// Mitsubishi GX Works2 project: PLC_GROUP17   PLC: FX3G

// global labels: Global1
VAR_GLOBAL
  work_day AT X007 : BOOL;
  active_day AT Y007 : BOOL;
  emergency_sw AT X005 : BOOL;
  enter_inventory AT X010 : BOOL;
  chocolate_stock AT D1100 : REAL;
  input_chocolate AT D1110 : REAL;
  nuts_stock AT D1120 : REAL;
  input_nuts AT D1130 : REAL;
  pistachio_stock AT D1140 : REAL;
  input_pistachio AT D1150 : REAL;
  kadaif_stock AT D1160 : REAL;
  input_kadaif AT D1170 : REAL;
  input_sw AT M0 : BOOL;
  check_stock AT M1 : BOOL;
  finish_one_pack AT Y005 : BOOL;
END_VAR
VAR_GLOBAL CONSTANT
  min_chocolate_stock : REAL := 400.0;
  min_nuts_stock : REAL := 100.0;
  min_pistachio : REAL := 120.0;
  min_kadaif_stock : REAL := 60.0;
END_VAR
VAR_GLOBAL
  chack_chocolate AT M2 : BOOL;
  check_choco AT M2 : BOOL;
  check_nuts AT M3 : BOOL;
  check_pist AT M4 : BOOL;
  check_kadaif AT M5 : BOOL;
  start_melting AT X001 : BOOL;
  melting_light AT Y001 : BOOL;
  sensor_45 AT X002 : BOOL;
END_VAR
VAR_GLOBAL CONSTANT
  choco_amount : REAL := 400.0;
END_VAR
VAR_GLOBAL
  location_sensor AT X003 : BOOL;
  casting_light AT Y002 : BOOL;
  casting_timer AT TC200 : BOOL;
END_VAR
VAR_GLOBAL CONSTANT
  cast_time : INT := 400;
END_VAR
VAR_GLOBAL
  end_casting AT TS200 : BOOL;
  end_cast_light AT M6 : BOOL;
  sample_type AT X004 : BOOL;
  analog_input1 AT D8280 : INT;
  save_analog_input AT D1180 : REAL;
END_VAR
VAR_GLOBAL CONSTANT
  max_for_mix_nuts : REAL := 5.0;
END_VAR
VAR_GLOBAL
  mix_nuts_approved AT M7 : BOOL;
  transfer_light AT M6 : BOOL;
END_VAR
VAR_GLOBAL CONSTANT
  const400 : REAL := 400.0;
  const100 : REAL := 100.0;
END_VAR
VAR_GLOBAL
  mix_dubai_approved AT M8 : BOOL;
END_VAR
VAR_GLOBAL CONSTANT
  const60 : REAL := 60.0;
  const120 : REAL := 120.0;
  const20 : REAL := 20.0;
END_VAR
VAR_GLOBAL
  start_filling AT M9 : BOOL;
  timer_5_sec AT TC210 : BOOL;
END_VAR
VAR_GLOBAL CONSTANT
  filling_time : INT := 500;
END_VAR
VAR_GLOBAL
  filling_timer AT TS210 : BOOL;
  blink1 AT TC1 : BOOL;
END_VAR
VAR_GLOBAL CONSTANT
  blink1_time : INT := 10;
END_VAR
VAR_GLOBAL
  blink2 AT TC11 : BOOL;
END_VAR
VAR_GLOBAL CONSTANT
  blink_time : INT := 5;
END_VAR
VAR_GLOBAL
  blink_timer2 AT TS11 : BOOL;
  blink_light AT M10 : BOOL;
  blink_light1 AT Y003 : BOOL;
  blink_timer1 AT TS1 : BOOL;
  blink_light2 AT Y004 : BOOL;
  start_kirur AT X006 : BOOL;
  kirur_timer AT TC21 : BOOL;
END_VAR
VAR_GLOBAL CONSTANT
  kirur_time : INT := 30;
END_VAR
VAR_GLOBAL
  end_kirur AT TS21 : BOOL;
  kirur_light AT Y006 : BOOL;
  pack_table AT X000 : BOOL;
  table_counter AT CC0 : BOOL;
END_VAR
VAR_GLOBAL CONSTANT
  const4 : INT := 4;
END_VAR
VAR_GLOBAL
  pact_table_light AT Y005 : BOOL;
  end_full_package AT CS0 : BOOL;
  storage AT D1190 : REAL;
END_VAR
VAR_GLOBAL CONSTANT
  const1 : REAL := 1.0;
  const10 : INT := 10;
END_VAR
VAR_GLOBAL
  output AT D8282 : INT;
  reset_light AT M11 : BOOL;
  hold AT M12 : BOOL;
  hold2 AT M13 : BOOL;
  hold3 AT M14 : BOOL;
END_VAR
VAR_GLOBAL CONSTANT
  const40 : REAL := 40.0;
END_VAR
VAR_GLOBAL
  reset_storage_light AT M15 : BOOL;
END_VAR
VAR_GLOBAL CONSTANT
  const0 : REAL;
  const00 : INT;
END_VAR
VAR_GLOBAL
  which_mix AT M16 : BOOL;
  choco_sub_light AT M17 : BOOL;
END_VAR

// task Task_01 (event TRUE, interval 0, priority 31): POU_01

PROGRAM POU_01
(* structured ladder/FBD written out as ST: instructions are called as NAME(EN, inputs, outputs); _pN, _eN, _tN stand for wires *)
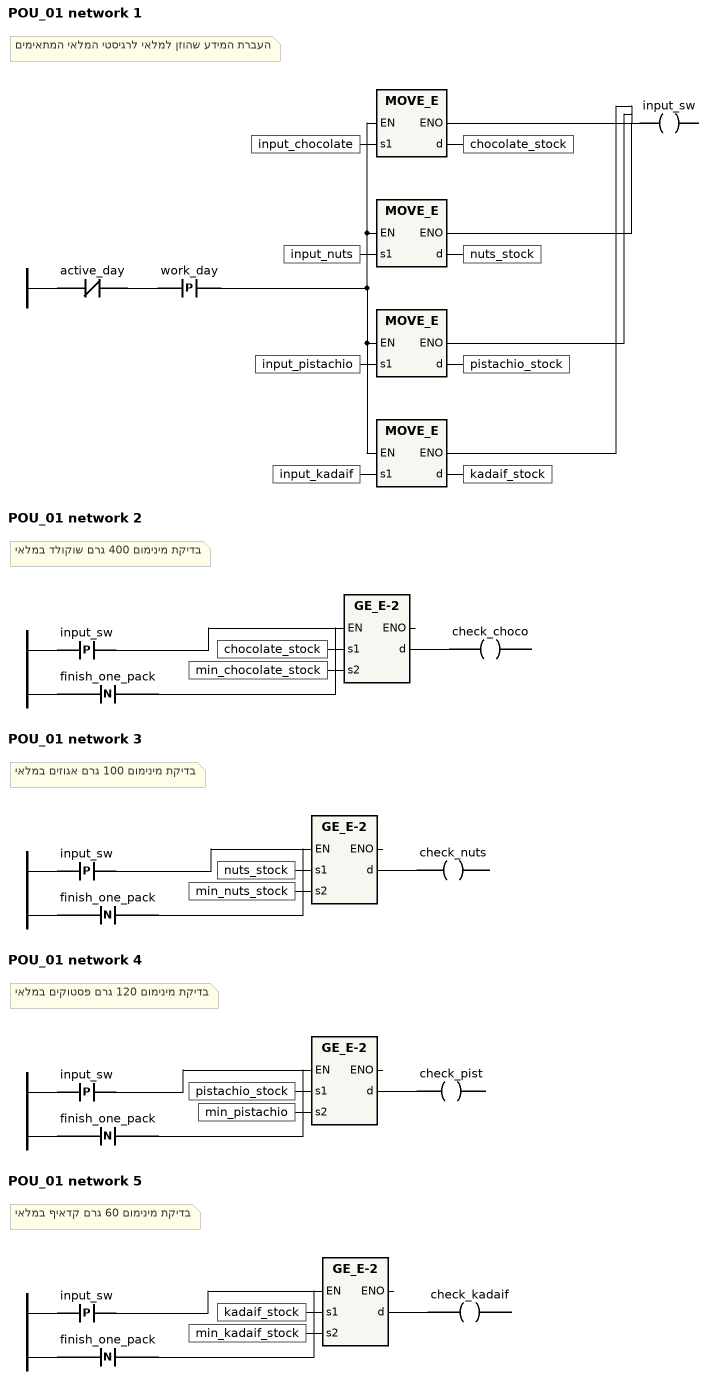
(* network 1 *)
(* העברת המידע שהוזן למלאי לרגיסטי המלאי המתאימים *)
_p1 := NOT active_day AND LDP(TRUE, work_day);
_e2 := MOVE_E(_p1, input_chocolate, chocolate_stock);
_e3 := MOVE_E(_p1, input_nuts, nuts_stock);
_e4 := MOVE_E(_p1, input_pistachio, pistachio_stock);
_e5 := MOVE_E(_p1, input_kadaif, kadaif_stock);
input_sw := _e2 OR _e3 OR _e4 OR _e5;
(* network 2 *)
(* בדיקת מינימום 400 גרם שוקולד במלאי *)
GE_E(LDP(TRUE, input_sw) OR LDF(TRUE, finish_one_pack), chocolate_stock, min_chocolate_stock, _t1);
check_choco := _t1;
(* network 3 *)
(* בדיקת מינימום 100 גרם אגוזים במלאי *)
GE_E(LDP(TRUE, input_sw) OR LDF(TRUE, finish_one_pack), nuts_stock, min_nuts_stock, _t1);
check_nuts := _t1;
(* network 4 *)
(* בדיקת מינימום 120 גרם פסטוקים במלאי *)
GE_E(LDP(TRUE, input_sw) OR LDF(TRUE, finish_one_pack), pistachio_stock, min_pistachio, _t1);
check_pist := _t1;
(* network 5 *)
(* בדיקת מינימום 60 גרם קדאיף במלאי *)
GE_E(LDP(TRUE, input_sw) OR LDF(TRUE, finish_one_pack), kadaif_stock, min_kadaif_stock, _t1);
check_kadaif := _t1;
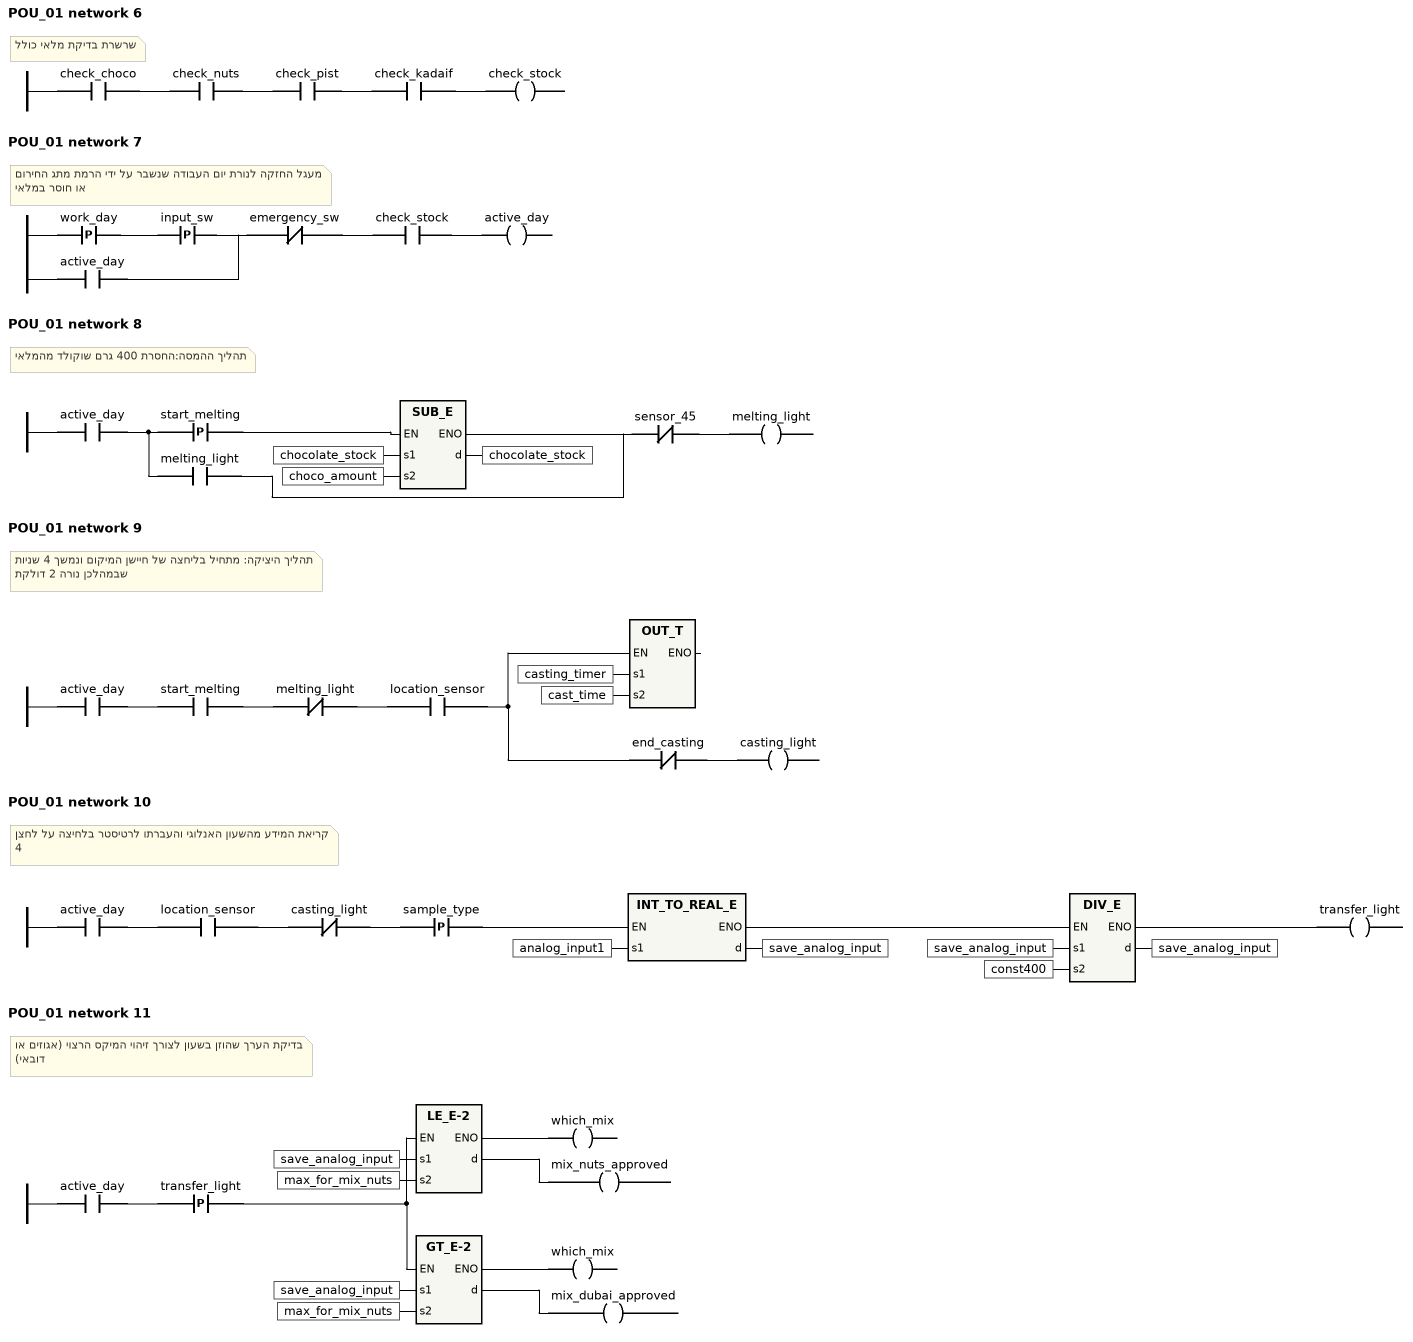
(* network 6 *)
(* שרשרת בדיקת מלאי כולל *)
check_stock := check_choco AND check_nuts AND check_pist AND check_kadaif;
(* network 7 *)
(* מעגל החזקה לנורת יום העבודה שנשבר על ידי הרמת מתג החירום או חוסר במלאי *)
active_day := (((LDP(TRUE, work_day) AND LDP(TRUE, input_sw)) OR active_day) AND NOT emergency_sw) AND check_stock;
(* network 8 *)
(* תהליך ההמסה:החסרת 400 גרם שוקולד מהמלאי *)
_e1 := SUB_E(active_day AND LDP(TRUE, start_melting), chocolate_stock, choco_amount, chocolate_stock);
melting_light := (_e1 OR (active_day AND melting_light)) AND NOT sensor_45;
(* network 9 *)
(* תהליך היציקה: מתחיל בליחצה של חיישן המיקום ונמשך 4 שניות שבמהלכן נורה 2 דולקת *)
_p1 := active_day AND start_melting AND NOT melting_light AND location_sensor;
OUT_T(_p1, casting_timer, cast_time);
casting_light := _p1 AND NOT end_casting;
(* network 10 *)
(* קריאת המידע מהשעון האנלוגי והעברתו לרטיסטר בלחיצה על לחצן 4 *)
_e1 := INT_TO_REAL_E(active_day AND location_sensor AND NOT casting_light AND LDP(TRUE, sample_type), analog_input1, save_analog_input);
_e2 := DIV_E(_e1, save_analog_input, const400, save_analog_input);
transfer_light := _e2;
(* network 11 *)
(* בדיקת הערך שהוזן בשעון לצורך זיהוי המיקס הרצוי (אגוזים או דובאי) *)
_p1 := active_day AND LDP(TRUE, transfer_light);
_e3 := LE_E(_p1, save_analog_input, max_for_mix_nuts, _t2);
which_mix := _e3;
mix_nuts_approved := _t2;
_e5 := GT_E(_p1, save_analog_input, max_for_mix_nuts, _t4);
which_mix := _e5;
mix_dubai_approved := _t4;
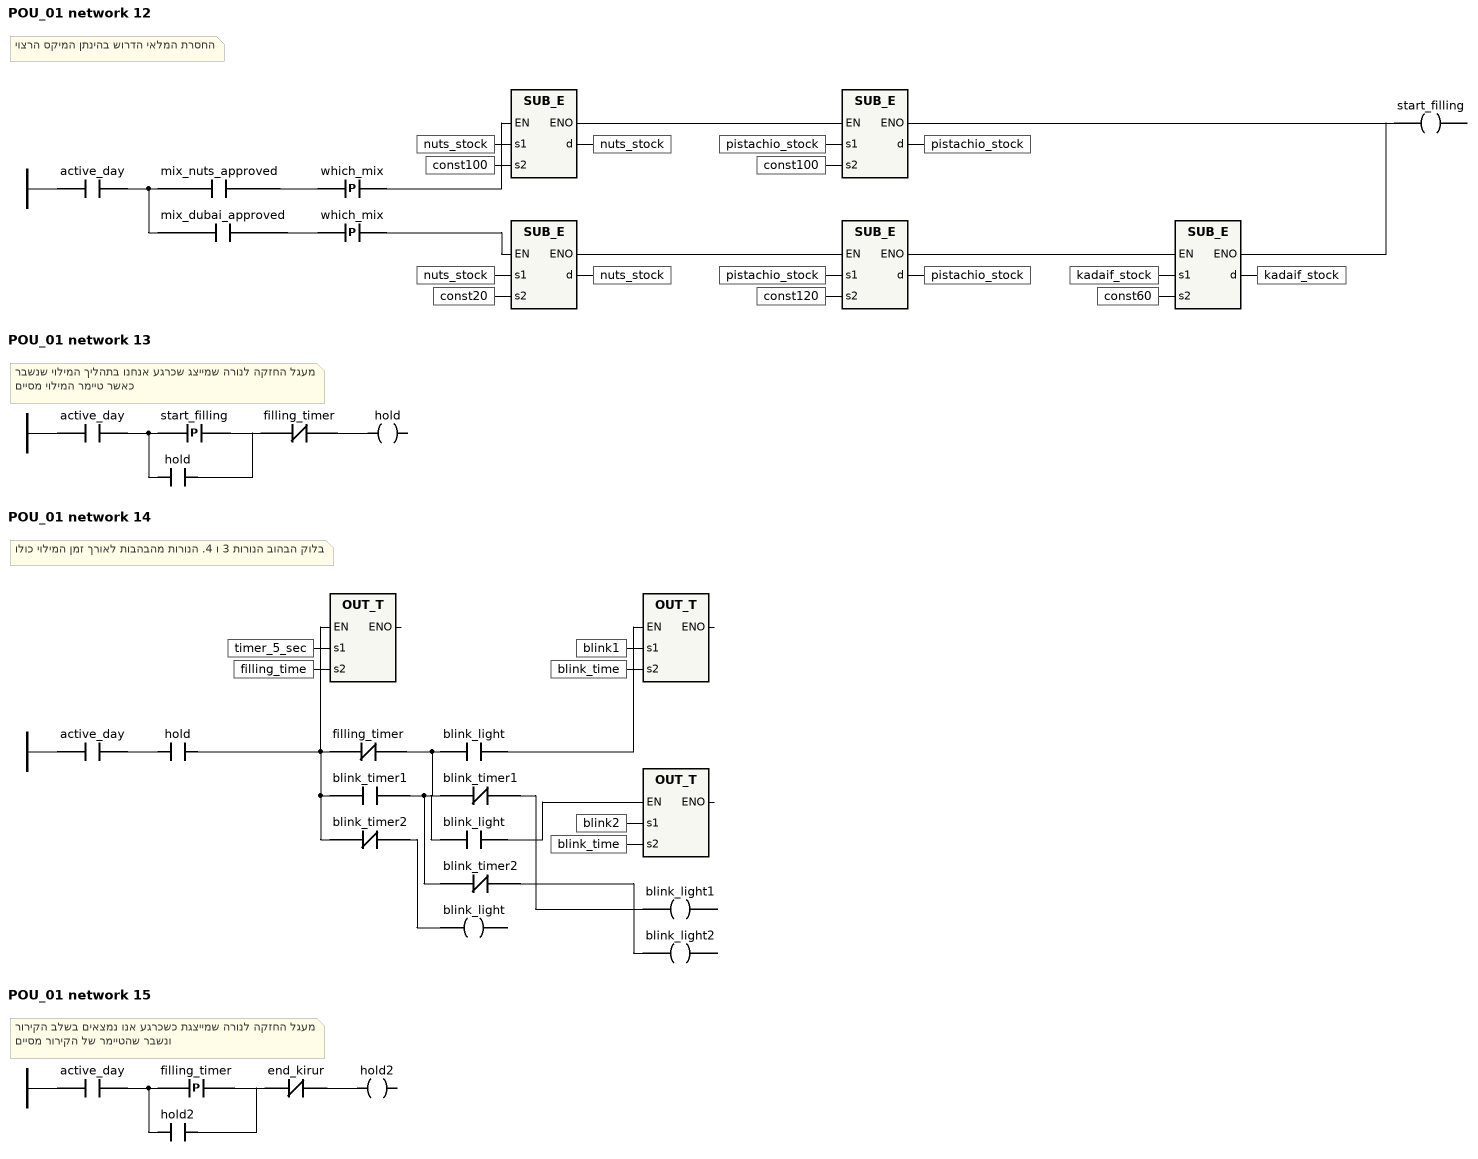
(* network 12 *)
(* החסרת המלאי הדרוש בהינתן המיקס הרצוי *)
_e1 := SUB_E(active_day AND mix_nuts_approved AND LDP(TRUE, which_mix), nuts_stock, const100, nuts_stock);
_e2 := SUB_E(_e1, pistachio_stock, const100, pistachio_stock);
_e3 := SUB_E(active_day AND mix_dubai_approved AND LDP(TRUE, which_mix), nuts_stock, const20, nuts_stock);
_e4 := SUB_E(_e3, pistachio_stock, const120, pistachio_stock);
_e5 := SUB_E(_e4, kadaif_stock, const60, kadaif_stock);
start_filling := _e2 OR _e5;
(* network 13 *)
(* מעגל החזקה לנורה שמייצג שכרגע אנחנו בתהליך המילוי שנשבר כאשר טיימר המילוי מסיים *)
hold := ((active_day AND LDP(TRUE, start_filling)) OR (active_day AND hold)) AND NOT filling_timer;
(* network 14 *)
(* בלוק הבהוב הנורות 3 ו 4. הנורות מהבהבות לאורך זמן המילוי כולו *)
_p1 := active_day AND hold;
OUT_T(_p1, timer_5_sec, filling_time);
_p2 := _p1 AND NOT filling_timer;
OUT_T(_p2 AND blink_light, blink1, blink_time);
blink_light1 := _p2 AND NOT blink_timer1;
_p3 := _p1 AND blink_timer1;
OUT_T(_p3 AND blink_light, blink2, blink_time);
blink_light2 := _p3 AND NOT blink_timer2;
blink_light := _p1 AND NOT blink_timer2;
(* network 15 *)
(* מעגל החזקה לנורה שמייצגת כשכרגע אנו נמצאים בשלב הקירור ונשבר שהטיימר של הקירור מסיים *)
hold2 := ((active_day AND LDP(TRUE, filling_timer)) OR (active_day AND hold2)) AND NOT end_kirur;
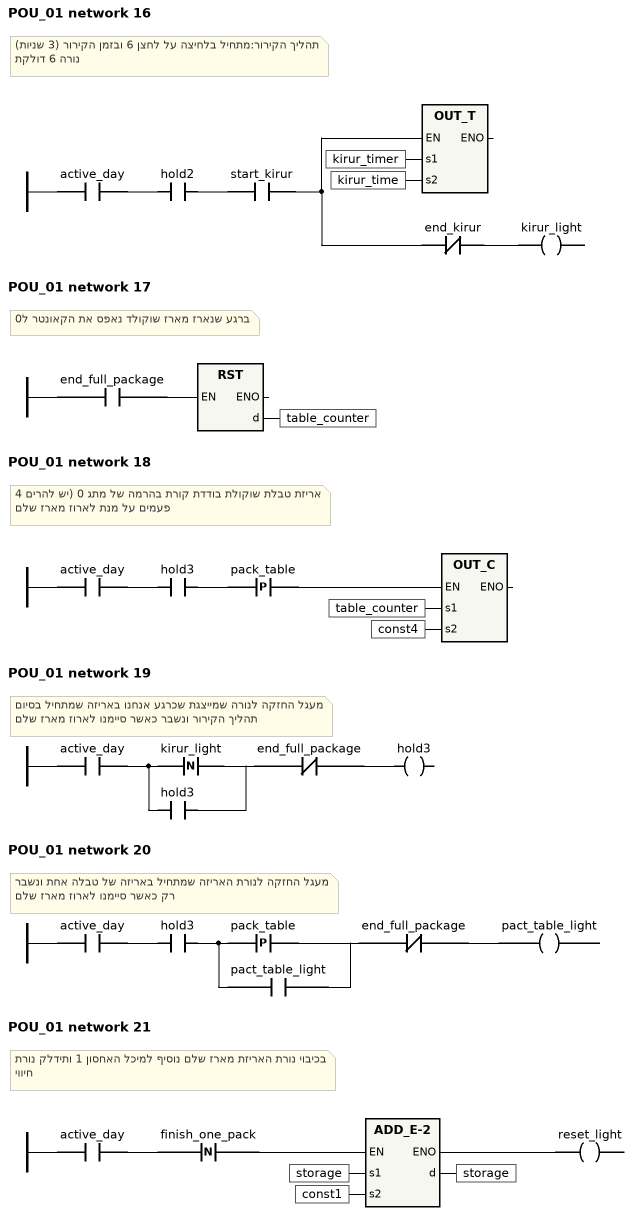
(* network 16 *)
(* תהליך הקירור:מתחיל בלחיצה על לחצן 6 ובזמן הקירור (3 שניות) נורה 6 דולקת *)
_p1 := active_day AND hold2 AND start_kirur;
OUT_T(_p1, kirur_timer, kirur_time);
kirur_light := _p1 AND NOT end_kirur;
(* network 17 *)
(* ברגע שנארז מארז שוקולד נאפס את הקאונטר ל0 *)
RST(end_full_package, table_counter);
(* network 18 *)
(* אריזת טבלת שוקולת בודדת קורת בהרמה של מתג 0 (יש להרים 4 פעמים על מנת לארוז מארז שלם *)
OUT_C(active_day AND hold3 AND LDP(TRUE, pack_table), table_counter, const4);
(* network 19 *)
(* מעגל החזקה לנורה שמייצגת שכרגע אנחנו באריזה שמתחיל בסיום תהליך הקירור ונשבר כאשר סיימנו לארוז מארז שלם *)
hold3 := ((active_day AND LDF(TRUE, kirur_light)) OR (active_day AND hold3)) AND NOT end_full_package;
(* network 20 *)
(* מעגל החזקה לנורת האריזה שמתחיל באריזה של טבלה אחת ונשבר רק כאשר סיימנו לארוז מארז שלם *)
_p1 := active_day AND hold3;
pact_table_light := ((_p1 AND LDP(TRUE, pack_table)) OR (_p1 AND pact_table_light)) AND NOT end_full_package;
(* network 21 *)
(* בכיבוי נורת האריזת מארז שלם נוסיף למיכל האחסון 1 ותידלק נורת חיווי *)
_e1 := ADD_E(active_day AND LDF(TRUE, finish_one_pack), storage, const1, storage);
reset_light := _e1;
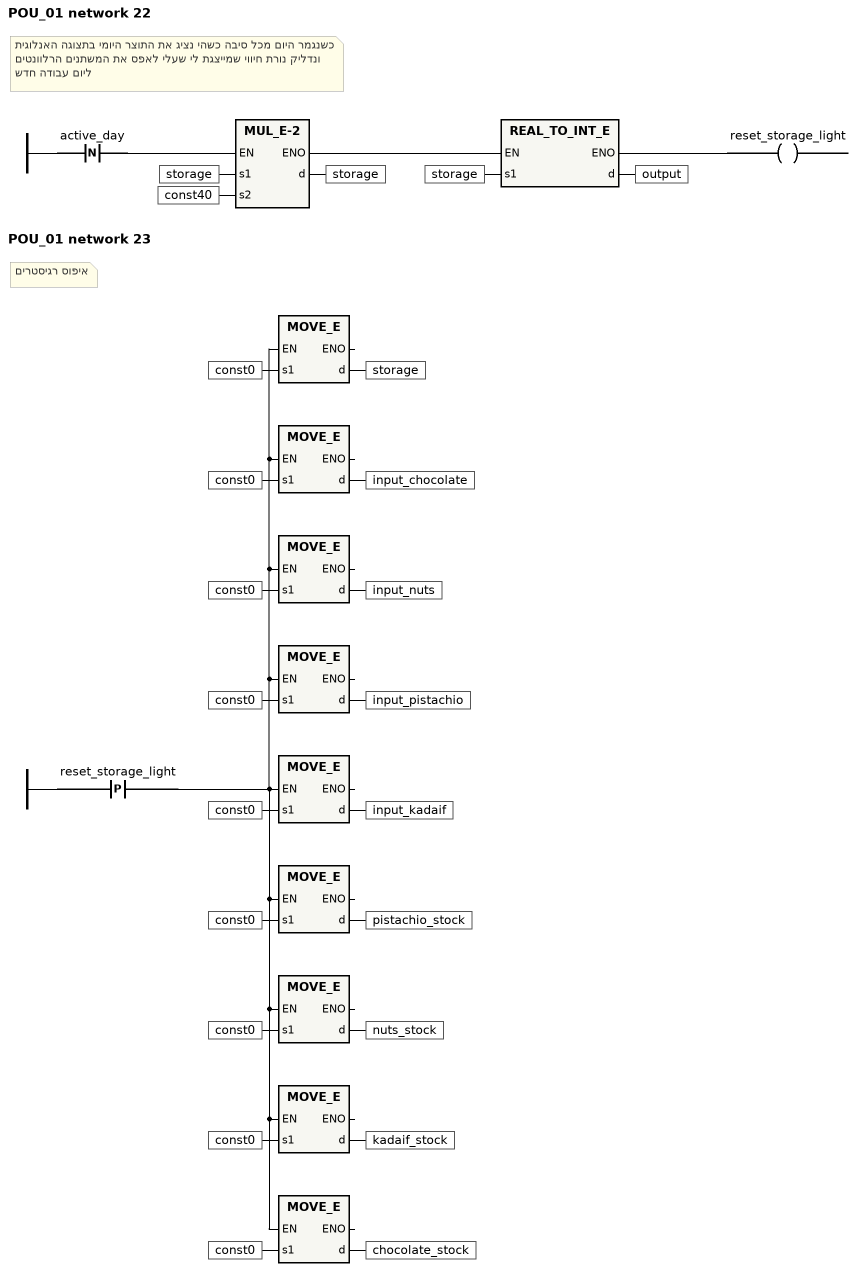
(* network 22 *)
(* כשנגמר היום מכל סיבה כשהי נציג את התוצר היומי בתצוגה האנלוגית ונדליק נורת חיווי שמייצגת לי שעלי לאפס את המשתנים הרלוונטים ליום עבודה חדש *)
_e1 := MUL_E(LDF(TRUE, active_day), storage, const40, storage);
_e2 := REAL_TO_INT_E(_e1, storage, output);
reset_storage_light := _e2;
(* network 23 *)
(* איפוס רגיסטרים *)
_p1 := LDP(TRUE, reset_storage_light);
MOVE_E(_p1, const0, storage);
MOVE_E(_p1, const0, input_chocolate);
MOVE_E(_p1, const0, input_nuts);
MOVE_E(_p1, const0, input_pistachio);
MOVE_E(_p1, const0, input_kadaif);
MOVE_E(_p1, const0, pistachio_stock);
MOVE_E(_p1, const0, nuts_stock);
MOVE_E(_p1, const0, kadaif_stock);
MOVE_E(_p1, const0, chocolate_stock);
END_PROGRAM
